// TIA Portal V18 export
TYPE "RCS_SysSafety_V1"
// stored: IsFailsafeCompliant false
   STRUCT
      LightCurtainOK : Array[0..7] of Bool;   // [0]=Total light curtain OK signal
      DoorClose : Array[0..15] of Bool;   // [0]=Total Safety door closed signal
      DoorLock : Array[0..15] of Bool;   // [0]=Total Safety door locked signal
      DoorOK : Array[0..15] of Bool;   // [0]=Total Safety door OK signal (Closed&Locked&be reset)
      DoorBypass : Bool;
   END_STRUCT;
END_TYPE
